PROGRAM prg_PWM
VAR
END_VAR

END_PROGRAM

(* stored: Version 1.1.0.1, ProductVersion 3.1.4024.15
   POU prg_PWM: Id {cb594440-59ea-46ee-beb4-c1d9f1bc6c1a}, SpecialFunc None *)
